TYPE (* A Structure with 2 Bits *)
  (* Version 1.0, 2024-02-21, franz *)
  st02b : STRUCT
    b00 : BOOL; (* BIT 00 *)
    b01 : BOOL; (* BIT 01 *)
  END_STRUCT;
END_TYPE
